// TIA Portal project "Lezione1_CorsoBase" (V19)

(* hardware
DEVICE "S7-1200 station_1"  S7-1200 Station
   slot 0: "Rack_0"  S7-1200 Rack  Rack  V1.0
   slot 1: "PLC_1"  CPU 1214C AC/DC/Rly  6ES7 214-1BG40-0XB0  V4.1
*)

// ===== PLC "PLC_1"  CPU 1214C AC/DC/Rly =====

VAR_GLOBAL   // PLC tag table "Default tag table"
   "PulsanteEmergenza" AT %I0.0 : Bool;
   "PulsanteStop" AT %I0.1 : Bool;
   "TermicaMotore" AT %I0.2 : Bool;
   "StartAvanti" AT %I0.3 : Bool;
   "StartIndietro" AT %I0.4 : Bool;
   "ResetAllarmi" AT %I0.5 : Bool;
   "ResetConteggio" AT %I0.6 : Bool;
   "MotoreAvanti" AT %Q0.0 : Bool;
   "MotoreIndietro" AT %Q0.1 : Bool;
   "LampadaVerde" AT %Q0.2 : Bool;
   "LampadaGialla" AT %Q0.3 : Bool;
   "LampadaRossa" AT %Q0.4 : Bool;
END_VAR

DATA_BLOCK "Motore1"   // DB1
{ S7_Optimized_Access := 'TRUE' }
VERSION : 0.1
// stored: InstanceOfName Motore
"Motore"
BEGIN
END_DATA_BLOCK

DATA_BLOCK "Motore2"   // DB2
{ S7_Optimized_Access := 'TRUE' }
VERSION : 0.1
// stored: InstanceOfName Motore
"Motore"
BEGIN
END_DATA_BLOCK

FUNCTION_BLOCK "Motore"   // FB1, LAD
{ S7_Optimized_Access := 'TRUE' }
VERSION : 0.1
   VAR_INPUT
      StartAvanti : Bool;
      StartIndietro : Bool;
      Stop : Bool;
      Termica : Bool;
      ResetAllarme : Bool;
      ResetConteggio : Bool;
   END_VAR
   VAR_OUTPUT
      MotoreAvanti : Bool;
      MotoreIndietro : Bool;
      StatoAttuale : Int;
   END_VAR
BEGIN
END_FUNCTION_BLOCK

ORGANIZATION_BLOCK "Main"   // OB1, LAD, ProgramCycle
TITLE = "Main Program Sweep (Cycle)"
{ S7_Optimized_Access := 'TRUE' }
VERSION : 0.1
   VAR_INPUT
      Initial_Call : Bool;   // Initial call of this OB
      Remanence : Bool;   // =True, if remanent data are available
   END_VAR
BEGIN

REGION Network 1
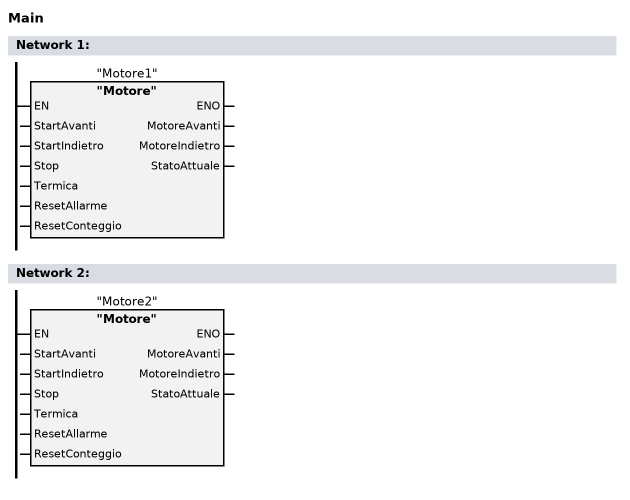
   RUNG wire#powerrail
      "Motore1"(StartAvanti :=, StartIndietro :=, Stop :=, Termica :=, ResetAllarme :=, ResetConteggio :=, MotoreAvanti =>, MotoreIndietro =>, StatoAttuale =>)
   END_RUNG
   // the same network as SCL:
   "Motore1"();   // "Motore"
END_REGION

REGION Network 2
   RUNG wire#powerrail
      "Motore2"(StartAvanti :=, StartIndietro :=, Stop :=, Termica :=, ResetAllarme :=, ResetConteggio :=, MotoreAvanti =>, MotoreIndietro =>, StatoAttuale =>)
   END_RUNG
   // the same network as SCL:
   "Motore2"();   // "Motore"
END_REGION
END_ORGANIZATION_BLOCK